TYPE ST_AxisPersistent :
STRUCT

    /////////Settings for restoring positions on power off/////////
    iPositionAtShutdown : LREAL;  //The position that the axis was at when CPU shut down
    bMovingAtShutdown   : BOOL;   //True if the axis was moving at shutdown, False otherwise 

END_STRUCT
END_TYPE

(* stored: Version 1.1.0.1, ProductVersion 3.1.4024.0
   DUT ST_AxisPersistent: Id {98d769cd-5416-4343-814a-f5a739d71156} *)
